INTERFACE I_OPCUA_Connect

METHOD start : BOOL
VAR_INPUT
    Execute            : BOOL;
    ServerUrl          : STRING(MAX_STRING_LENGTH);
    SessionConnectInfo : ST_UASessionConnectInfo;     
    Timeout            : TIME := DEFAULT_ADS_TIMEOUT; 
END_VAR
VAR_OUTPUT
    ConnectionHdl : DWORD;
    Done          : BOOL;
    Busy          : BOOL;
    Error         : BOOL;
    ErrorID       : DWORD;
END_VAR
END_METHOD

END_INTERFACE

(* stored: Version 1.1.0.1, ProductVersion 3.1.4024.9
   Itf I_OPCUA_Connect: Id {6a688e78-a1c4-438f-a51a-56d256578318}
   Method start: Id {35e2e35e-ec82-4e4a-bcbe-c76ff647fb80} *)
